Fanuc KAREL source: kb00060.KL

PROGRAM KB00060
%NOLOCKGROUP
VAR
P1 : STRING[80];P2:INTEGER;P3:INTEGER;P4:INTEGER;P5:INTEGER
BEGIN
--
--
--
--
P1='A'
P2=1
P3=1
P4=1
P5=1
DEF_WINDOW(P1,P2,P3,P4,P5)
END KB00060
